FUNCTION_BLOCK AxisDisableCommand IMPLEMENTS ITF_Command
VAR
END_VAR

{warning 'add method implementation '}
METHOD Execute : BOOL
END_METHOD

END_FUNCTION_BLOCK

(* stored: Version 1.1.0.1, ProductVersion 3.1.4024.12
   POU AxisDisableCommand: Id {2a2d0b49-8a40-4eea-91a3-a3f65d5fce60}, SpecialFunc None
   Method Execute: Id {35963484-04dd-45ff-b5c9-11e500c894f5} *)
